PROGRAM P_counter
VAR
	iCounter : INT := 0;
END_VAR

iCounter := iCounter +1;

END_PROGRAM

(* stored: Version 1.1.0.1, ProductVersion 3.1.4024.9
   POU P_counter: Id {83c85a13-f4ab-43fb-b683-b335d8183aae}, SpecialFunc None *)
